Staubli VAL3: goTo.pgx

public program goTo(tool x_tTool, mdesc x_mDesc, num x_nMoveType, bool& x_bUnreached[], num x_nIndex)
  local point l_pTrsf
  local bool l_bInside
  local tool l_tTool
  local point l_pHere
  local string l_sMessage
  local num l_nSize
  local num i
begin
  // the maximum size
  if isInRange(jEditPoint.tData[x_nIndex].jJoint)
    // go to the select Joint
    movej(jEditPoint.tData[x_nIndex].jJoint,x_tTool,x_mDesc)
  else
    x_bUnreached=true
  endIf
end
